TYPE EL3xx2_Data :
STRUCT
	{attribute addProperty Name "AI Standard Channel 1"}
	_1 : AI_Standard_Channel;
	{attribute addProperty Name "AI Standard Channel 2"}
	_2 : AI_Standard_Channel;
END_STRUCT
END_TYPE

(* stored: Version 1.1.0.1, ProductVersion 3.1.4024.9
   DUT EL3xx2_Data: Id {d417c3e7-abd8-05ba-29c6-2191cad4362e} *)
